FUNCTION_BLOCK LopendeBand implements ITFMotor
VAR_INPUT
END_VAR
VAR_OUTPUT
END_VAR
VAR
END_VAR

// kan aan en uit en reageert op errors, heeft lichtsensor aan het einde van het banddel

METHOD HandleErrors : BOOL
VAR_INPUT
END_VAR
END_METHOD

METHOD LichtSensor : BOOL
VAR_INPUT
END_VAR
END_METHOD

PROPERTY LopendeBandStatus : ELopendeBandStatus
GET
END_GET
SET
END_SET
END_PROPERTY

METHOD MotorAan
VAR_INPUT
END_VAR
END_METHOD

METHOD MotorUit
VAR_INPUT
END_VAR
END_METHOD

END_FUNCTION_BLOCK

(* stored: Version 1.1.0.1
   POU LopendeBand: Id {af1489a2-4b96-41ec-9023-dbc3371340a0}, SpecialFunc None
   Method HandleErrors: Id {4482d789-05c3-4af2-9881-523428224908}
   Method LichtSensor: Id {e295db0b-e309-4826-aa12-b8844bc13c3f}
   Property LopendeBandStatus: Id {e25f0d20-e450-4241-b528-fbcd05cd4bf1}
   Get Get: Id {7bf1af54-c934-41f2-97ee-94bf6422b8bf}
   Set Set: Id {89f06e9d-0dbc-4bb0-9d04-ba961ffc06be}
   Method MotorAan: Id {9103c7af-6c47-4658-92d4-6ad86d23e3a9}
   Method MotorUit: Id {6cf8c88b-0239-4171-9cdc-4661629a3699} *)
